Staubli VAL3: doTest.pgx

program doTest()
begin
  call park1()

  while true

    if bDoTest==true
      if statusValves[hdiValve[0]]==0 or statusValves[sensorValve[0]]==0
        userPageAlert("No vaccum applied to airex #0. Fix this first!")
        return
      elseIf statusValves[hdiValve[1]]==0
        userPageAlert("No vaccum applied to airex #1. Fix this first!")
        return
      elseIf statusValves[hdiValve[2]]==0
        userPageAlert("No vaccum applied to airex #2. Fix this first!")
        return
      elseIf statusValves[hdiValve[3]]==0
        userPageAlert("No vaccum applied to airex #3. Fix this first!")
        return
      elseIf statusValves[hdiValve[4]]==0
        userPageAlert("No vaccum applied to airex #4. Fix this first!")
        return
      elseIf statusValves[hdiValve[5]]==0
        userPageAlert("No vaccum applied to airex #5. Fix this first!")
        return
      endIf
    endIf

  endWhile
end
